# B&R Automation Studio project laba1
Automation Studio 4.5.2.102

## Configuration Config1

### Task classes (Cpu.sw)
```
Cyclic#4:
  Program <- Program.prg
Libraries: MotorCha
```

### Hardware
```
4PP065_0571_P74 : 4PP065.0571-P74 v1.1.2.0
  Connector IF5:
    ActivateDevice = 1
  ConfigurationID = lab11_Config1
  Simulation = 1
```

## Logical view

Binary libraries used (declarations not repeated): operator, runtime, astime, AsIecCon

### Global.var
```iecst
VAR
	New_Variable : USINT;
END_VAR
```

### Library Logical/Libraries/MotorCha (ANSIC)

#### Constants.var - Exported constants
```iecst
VAR CONSTANT
	delta_t : REAL := 0.01;
END_VAR
```

#### MotorCha.fun - Exported functions and function blocks
```iecst
{REDUND_ERROR} {REDUND_UNREPLICABLE} FUNCTION_BLOCK FB_Integrator (*TODO: Add your comment here*) (*$GROUP=User,$CAT=User,$GROUPICON=User.png,$CATICON=User.png*)
	VAR_INPUT
		in : {REDUND_UNREPLICABLE} REAL;
	END_VAR
	VAR_OUTPUT
		out : {REDUND_UNREPLICABLE} REAL;
	END_VAR
	VAR
		dt : {REDUND_UNREPLICABLE} REAL;
		prev_value : {REDUND_UNREPLICABLE} REAL;
	END_VAR
END_FUNCTION_BLOCK

{REDUND_ERROR} FUNCTION_BLOCK FB_Motor (*TODO: Add your comment here*) (*$GROUP=User,$CAT=User,$GROUPICON=User.png,$CATICON=User.png*)
	VAR_INPUT
		u : {REDUND_UNREPLICABLE} REAL;
	END_VAR
	VAR_OUTPUT
		w : {REDUND_UNREPLICABLE} REAL;
		phi : {REDUND_UNREPLICABLE} REAL;
	END_VAR
	VAR
		integrator : {REDUND_UNREPLICABLE} FB_Integrator;
		Tm : {REDUND_UNREPLICABLE} REAL := 0.04;
		ke : {REDUND_UNREPLICABLE} REAL := 208.33;
		dt : {REDUND_UNREPLICABLE} REAL;
		prev_value : REAL;
	END_VAR
END_FUNCTION_BLOCK

{REDUND_ERROR} FUNCTION_BLOCK FB_Regulator (*TODO: Add your comment here*) (*$GROUP=User,$CAT=User,$GROUPICON=User.png,$CATICON=User.png*)
	VAR_INPUT
		e : {REDUND_UNREPLICABLE} REAL;
	END_VAR
	VAR_OUTPUT
		u : {REDUND_UNREPLICABLE} REAL;
	END_VAR
	VAR
		k_p : {REDUND_UNREPLICABLE} REAL := 0.0064;
		integrator : {REDUND_UNREPLICABLE} FB_Integrator;
		k_i : {REDUND_UNREPLICABLE} REAL := 0.16;
		max_abs_value : {REDUND_UNREPLICABLE} REAL := 24;
		dt : {REDUND_UNREPLICABLE} REAL;
		last_sum : REAL;
		sum : REAL;
	END_VAR
END_FUNCTION_BLOCK
```

#### FB_Integrator.c
```c
#include <bur/plctypes.h>
#ifdef __cplusplus
	extern "C"
	{
#endif
	#include "MotorCha.h"
#ifdef __cplusplus
	};
#endif
/* TODO: Add your comment here */
void FB_Integrator(struct FB_Integrator* inst)
{
	inst->dt = delta_t;
	inst->out = inst->dt * inst->in + inst->prev_value;
	inst->prev_value = inst->out;
}
```

#### FB_Motor.c
```c
#include <bur/plctypes.h>
#ifdef __cplusplus
	extern "C"
	{
#endif
	#include "MotorCha.h"
#ifdef __cplusplus
	};
#endif
/* TODO: Add your comment here */
void FB_Motor(struct FB_Motor* inst)
{
	REAL a = inst->u / inst->ke - inst->w;
	REAL b = a / inst->Tm;

	inst->integrator.in = b;
	FB_Integrator(&inst->integrator);

	inst->w = inst->integrator.out;
}
```

#### FB_Regulator.c
```c
#include <bur/plctypes.h>
#ifdef __cplusplus
	extern "C"
	{
#endif
	#include "MotorCha.h"
#ifdef __cplusplus
	};
#endif
/* TODO: Add your comment here */
void FB_Regulator(struct FB_Regulator* inst)
{
	REAL a = inst->e * inst->k_p;
	REAL b = inst->e * inst->k_i;

	a = a > inst->max_abs_value ? inst->max_abs_value : a;
	a = a < -inst->max_abs_value ? -inst->max_abs_value : a;

	inst->integrator.in = b + inst->last_sum;
	FB_Integrator(&inst->integrator);

	REAL sum = a + inst->integrator.out;

	inst->u = sum;
	inst->u = inst->u > inst->max_abs_value ? inst->max_abs_value : inst->u;
	inst->u = inst->u < -inst->max_abs_value ? -inst->max_abs_value : inst->u;

	inst->last_sum = inst->u - sum;
}
```

### Program Logical/Program

#### Variables.var
```iecst
VAR
	fb_controller : {REDUND_UNREPLICABLE} FB_Regulator;
	fb_motor1 : FB_Motor;
	fb_motor2 : FB_Motor;
	speed : REAL;
	counter : UINT;
	enable : BOOL;
END_VAR
```

#### Cyclic.c
```c
#include <bur/plctypes.h>

#ifdef _DEFAULT_INCLUDES
	#include <AsDefault.h>
#endif

void _CYCLIC ProgramCyclic(void)
{
	if(enable) {
		if(counter == 200) {
			speed = 0;
			counter = 0;
		}
		if(counter == 50) {
			speed = 50;
		}

		counter++;

		fb_controller.e = speed - fb_motor1.w;
		FB_Regulator(&fb_controller);
		fb_motor1.u = fb_controller.u;

		FB_Motor(&fb_motor1);

		fb_motor2.u = speed * fb_motor2.ke;
		FB_Motor(&fb_motor2);
	}
}
```

#### Init.c
```c
#include <bur/plctypes.h>

#ifdef _DEFAULT_INCLUDES
	#include <AsDefault.h>
#endif

void _INIT ProgramInit(void)
{
	speed = 0;
	counter = 0;
	enable = 0;
}
```

Listed in the project but not available here: Logical/Libraries/MotorCha/Types.typ
